(* IEC 61131-3 sources: CodesysTest/alpha/export/ElectricMachine.dev/Plc Logic/Application/Event Handlers, 2 files *)

(* ---- PrepareExitTasks.pou.st ---- *)
(*#-#-#-#-#-#-#-#-#-#---Declaration---#-#-#-#-#-#-#-#-#-#-#-#-#*)

FUNCTION PrepareExitTasks : DWORD
VAR_IN_OUT
	EventPrm: Component_Manager.EVTPARAM_CmpMgr_Shutdown;
END_VAR
VAR
END_VAR
(*#-#-#-#-#-#-#-#-#-#---Implementation---#-#-#-#-#-#-#-#-#-#-#-#-#*)

SaveValuesTest();

(* ---- PrepareShutdown.pou.st ---- *)
(*#-#-#-#-#-#-#-#-#-#---Declaration---#-#-#-#-#-#-#-#-#-#-#-#-#*)

FUNCTION PrepareShutdown : DWORD
VAR_IN_OUT
	EventPrm: Component_Manager.EVTPARAM_CmpMgr_Shutdown;
END_VAR
VAR
END_VAR
(*#-#-#-#-#-#-#-#-#-#---Implementation---#-#-#-#-#-#-#-#-#-#-#-#-#*)

SaveValues();
